//==================================================================================================
//							Beckhoff Automation Poland
//									3.01.2023
//	Function block running home procedure in torque mode detection
//	It doesn't change position - only detection implemented
//	lrRecordedPosition - catched position. Offset can be written i.e. to encoder memory
//
//	Avaliable two modes:
//	1. Lag based - bLagBased = TRUE - define lrLagLimit which decides about end of movement
//	2. Torque based - bLagBased = FALSE - define lrTorqueLimit and lrTorqueTolerance which decides about end of movement
//
//	Library: Tc3_MC2_AdvancedHoming, Tc2_MC2, 
//
//  v1.1	|| TC v 3.1.4024.35		|| Naming convention 
//  v1.0	|| TC v 3.1.4024.22		|| First edition 
//==================================================================================================
FUNCTION_BLOCK FB_HomingTorqueDetection
VAR_IN_OUT
	Axis 										: Tc2_MC2.AXIS_REF;
END_VAR  
VAR_INPUT
	bExecute									: BOOL;					// The command is executed with a rising edge.
	bLagBased									: BOOL;					// TRUE: MC_StepBlockLagBased, FALSE: MC_StepBlock
	eDirection									: Tc3_MC2_AdvancedHoming.MC_Home_Direction;	// 
	fVelocity									: LREAL;				// Maximum travel velocity (>0)
	fDetectionVelocityLimit						: LREAL;				// Velocity that must be fallen below for the time DetectionVelocityTime in order to detect driving against the fixed stop.
	tDetectionVelocityTime						: TIME;					// Time for detecting the velocity undershoot when driving against the fixed stop.
	tTimeLimit									: TIME;					// Exceeding this time leads to the search procedure being aborted.
	fDistanceLimit								: LREAL;				// Exceeding this distance in relation to the start position leads to the search procedure being aborted.
	fTorqueLimit								: LREAL;				// The motor torque is limited to this value, in relation to the weight counterbalance that is possibly parameterized in the drive, in order to avoid mechanical damage.
	fTorqueTolerance							: LREAL;				// Tolerance related to the TorqueLimit within which driving against the fixed stop is detected.
	fLagLimit									: LREAL;				// Position lag value which, if exceeded, leads to detection of driving against the fixed stop.
	fDistance									: LREAL;				// Distance by which the axis moves away from the current position.
END_VAR                             		
VAR_OUTPUT                              		
	bDone										: BOOL;
	bBusy										: BOOL;
	bCommandAborted								: BOOL;
	bError										: BOOL;
	nErrorID									: UDINT;
	fRecordedPosition							: LREAL;				// Catched position. Offset can be written i.e. to encoder memory
END_VAR
VAR
//=========================== Common ============================
	nStep										: DINT;
	stParameter									: Tc3_MC2_AdvancedHoming.MC_HomingParameter;
	stOptions									: Tc3_MC2_AdvancedHoming.ST_Home_Options3;
//========================= Step Block ==========================
	mcStepBlock									: Tc3_MC2_AdvancedHoming.MC_StepBlockDetection ;
	mcStepBlockLag								: Tc3_MC2_AdvancedHoming.MC_StepBlockLagBasedDetection;
//====================== Move Relative ==========================
	mcMoveRelative								: MC_MoveRelative;
//============================ Abort ============================
	mcAbortHoming								: Tc3_MC2_AdvancedHoming.MC_AbortHoming;
//========================== Internal ===========================
    {attribute 'hide'}
	nErrorID_Int								: UDINT;
//===============================================================
END_VAR

//====== Call FBs outside CASE - easier debugging ===============
mcStepBlockLag(Axis								:= Axis, 
				Parameter						:= stParameter);
				                        		
mcStepBlock(	Axis							:= Axis, 
				Parameter						:= stParameter);	

mcMoveRelative(	Axis							:= Axis);
                                        		
mcAbortHoming(	Axis							:= Axis, 
				Parameter						:= stParameter);
			
//============== CASE instruction - step machine ================
CASE nStep OF
	
	0: // Wait for command
	
		IF bExecute THEN
			bBusy								:= TRUE;
			// Latch finish parameters
			mcMoveRelative.Distance				:= fDistance;
			mcMoveRelative.Velocity				:= fVelocity;
			
			IF bLagBased THEN

				mcStepBlockLag(Axis				:= Axis, 
						Parameter				:= stParameter, 
						Execute					:= TRUE, 
						Direction				:= eDirection, 
						Velocity				:= fVelocity,
						DetectionVelocityLimit	:= fDetectionVelocityLimit, 
						DetectionVelocityTime	:= tDetectionVelocityTime, 
						TimeLimit				:= tTimeLimit, 
						DistanceLimit			:= fDistanceLimit, 
						TorqueLimit				:= fTorqueLimit, 
						LagLimit				:= fLagLimit, 
						Options					:= stOptions);
				
				nStep							:= 1000;
				
			ELSE

				mcStepBlock(Axis				:= Axis, 
						Parameter				:= stParameter, 
						Execute					:= TRUE, 
						Direction				:= eDirection, 
						Velocity				:= fVelocity,
						DetectionVelocityLimit	:= fDetectionVelocityLimit, 
						DetectionVelocityTime	:= tDetectionVelocityTime, 
						TimeLimit				:= tTimeLimit, 
						DistanceLimit			:= fDistanceLimit, 
						TorqueLimit				:= fTorqueLimit, 
						TorqueTolerance			:= fTorqueTolerance, 
						Options					:= stOptions);
						
				nStep							:= 2000;
				
			END_IF
		END_IF
	
	1000: // Wait till end MC_StepBlockLagBasedDetection
	
		IF mcStepBlockLag.Done THEN
			fRecordedPosition					:= mcStepBlockLag.RecordedPosition;
			mcStepBlockLag.Execute				:= FALSE;
			nStep 								:= 3000;
		END_IF
		
		IF mcStepBlockLag.CommandAborted THEN
			mcStepBlockLag.Execute				:= FALSE;
			nStep 								:= 6010;
		END_IF
		
		IF mcStepBlockLag.Error THEN
			mcStepBlockLag.Execute				:= FALSE;
			nErrorID_Int						:= mcStepBlockLag.ErrorID;
			nStep 								:= 6110;
		END_IF
	
	2000: // Wait till end MC_StepBlockDetection
	
		IF mcStepBlock.Done THEN
			fRecordedPosition					:= mcStepBlock.RecordedPosition;
			mcStepBlock.Execute					:= FALSE;
			nStep 								:= 3000;
		END_IF
		
		IF mcStepBlock.CommandAborted THEN
			mcStepBlock.Execute					:= FALSE;
			nStep 								:= 6020;
		END_IF
		
		IF mcStepBlock.Error THEN
			mcStepBlock.Execute					:= FALSE;
			nErrorID_Int						:= mcStepBlock.ErrorID;
			nStep 								:= 6120;
		END_IF
		
	3000:	// MC_AbortHoming - way of finish homing procedure
	
		mcAbortHoming.Execute					:= TRUE;				
		nStep									:= nStep + 10;
		
	3010: // Wait till end MC_HomeDirect
	
		IF mcAbortHoming.Done THEN
			mcAbortHoming.Execute				:= FALSE;
			nStep 								:= 4000;
		END_IF
		
		IF mcAbortHoming.CommandAborted THEN
			mcAbortHoming.Execute				:= FALSE;
			nStep 								:= 6040;
		END_IF
		
		IF mcAbortHoming.Error THEN
			mcAbortHoming.Execute				:= FALSE;
			nErrorID							:= mcAbortHoming.ErrorID;
			nStep 								:= 6140;
		END_IF		

	4000: // MC_MoveRelative
	
		mcMoveRelative.Execute					:= TRUE;			
		nStep									:= nStep + 10;
	
	4010: // Wait till end MC_MoveRelative
	
		IF mcMoveRelative.Done THEN
			mcMoveRelative.Execute				:= FALSE;
			bBusy 								:= FALSE;
			bDone 								:= TRUE;
			nStep								:= 5000;
		END_IF
		
		IF mcMoveRelative.CommandAborted THEN
			mcMoveRelative.Execute				:= FALSE;
			nStep 								:= 6050;
		END_IF
		
		IF mcMoveRelative.Error THEN
			mcMoveRelative.Execute				:= FALSE;
			nErrorID_Int						:= mcMoveRelative.ErrorID;
			nStep 								:= 6150;
		END_IF		
	
	5000: // Done
	
		bDone									:= bExecute;
		IF NOT bExecute THEN
			fRecordedPosition					:= 0;
			nStep 								:= 0;
		END_IF
	
	6000..6199: // MC_AbortHoming
	
		mcAbortHoming.Execute					:= TRUE;				
		nStep									:= nStep + 200;
	
	6200..6399: // Wait till end Command Aborted (..200-..299)/Error (..300/399)
	
		// No matter what is the end, we go to Command Aborted/Error State
		IF NOT mcAbortHoming.Busy THEN
			mcAbortHoming.Execute				:= FALSE;
			bBusy 								:= FALSE;
			// Set CA/E flag
			bCommandAborted						:= nStep < 6300;
			bError								:= NOT bCommandAborted;
			
			IF bError THEN
				nErrorID						:= nErrorID_Int;
				nStep							:= nStep + 10000;
			ELSE
				nStep							:= 7000;
			END_IF
		
		END_IF		
	
	7000: // Command Aborted
	
		bCommandAborted							:= bExecute;
		IF NOT bExecute THEN
			nStep 								:= 0;
		END_IF
		
	10000..20000: // Error
	
		bError									:= bExecute;
		IF NOT bExecute THEN
			nErrorID							:= 0;
			nErrorID_Int						:= 0;
			nStep 								:= 0;
		END_IF
		
END_CASE
//===============================================================

END_FUNCTION_BLOCK

(* stored: Version 1.2.0.0, ProductVersion 3.1.4026.13, FileIdentifier a144b101fe0b8aeb7822292b9dc0dd792c579fe0, FileSignature 8bf6f5bbcf6b199439564678508831c0f12a936a28f333c7e35e57667e326ed7fb436e8682b12855e958ff03d4cf329b38f1ec7ebbaf7c310d204a3013919a132a5113c633fe621c89848d9949705cc4b851a4eb8670aefc189e4ad6c2b237a5287e0a35ae698b93ef4f047a1b0aad3a497724a0e183610ea1daeeb8ec44db2b187624e25eb4f9a44a20f8441ea97bc1aad5e43edd9177bfdf55cc3ff74e3d459655760d983a7d6b13dc0df041d4f60053da92bd949c47e4ca105234306e80d41cc76a1fe7a58b4b48e15df4d4555728b67002a77be6f1d00812eb68de6b905beb510bf264d3b8d5295b3808b07f7bd6ce33fa9a30f3e73bc1d74204d1dbf5c5
   POU FB_HomingTorqueDetection: Id {787bcb89-acd4-4316-8722-98b052dee456}, SpecialFunc None *)
